SUBAPPLICATION Uebung_002a5b_AX (* DigitalInput_I1-3 mit OR auf DigitalOutput_Q1-3, mit Plug and Socket *)
  (* Standard: 61499-2; Description: Copyright (c) 2023 Meisterschulen am Ostbahnhof This program and the accompanying materials are made available under the terms of the Eclipse Public License 2.0 which is available at https://www.eclipse.org/legal/epl-2.0/ SPDX-License-Identifier: EPL-2.0 *)
  (* Version 1.0, 2023-10-23, Franz Höpfinger, Meisterschulen am Ostbahnhof, initial API and implementation and/or initial documentation *)
  PACKAGE Uebungen;
  IMPORT logiBUS::io::DI::logiBUS_DI::Input_I1;
  IMPORT logiBUS::io::DI::logiBUS_DI::Input_I2;
  IMPORT logiBUS::io::DI::logiBUS_DI::Input_I3;
  IMPORT logiBUS::io::DQ::logiBUS_DO::Output_Q1;
  IMPORT logiBUS::io::DQ::logiBUS_DO::Output_Q2;
  IMPORT logiBUS::io::DQ::logiBUS_DO::Output_Q3;
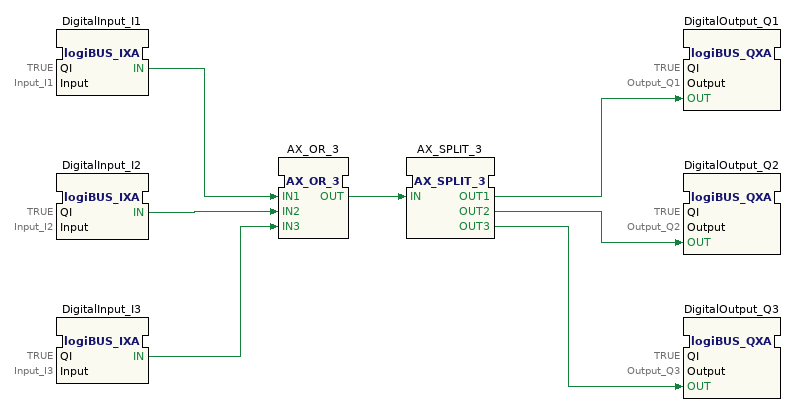
  FBS
    DigitalInput_I1 : logiBUS::io::DI::logiBUS_IXA(QI := TRUE, Input := Input_I1);
    DigitalOutput_Q1 : logiBUS::io::DQ::logiBUS_QXA(QI := TRUE, Output := Output_Q1);
    AX_OR_3 : adapter::booleanOperators::AX_OR_3;
    DigitalInput_I2 : logiBUS::io::DI::logiBUS_IXA(QI := TRUE, Input := Input_I2);
    DigitalInput_I3 : logiBUS::io::DI::logiBUS_IXA(QI := TRUE, Input := Input_I3);
    DigitalOutput_Q2 : logiBUS::io::DQ::logiBUS_QXA(QI := TRUE, Output := Output_Q2);
    DigitalOutput_Q3 : logiBUS::io::DQ::logiBUS_QXA(QI := TRUE, Output := Output_Q3);
    AX_SPLIT_3 : adapter::events::unidirectional::AX_SPLIT_3;
  END_FBS
  ADAPTER_CONNECTIONS
    DigitalInput_I1.IN TO AX_OR_3.IN1;
    DigitalInput_I2.IN TO AX_OR_3.IN2;
    DigitalInput_I3.IN TO AX_OR_3.IN3;
    AX_OR_3.OUT TO AX_SPLIT_3.IN;
    AX_SPLIT_3.OUT1 TO DigitalOutput_Q1.OUT;
    AX_SPLIT_3.OUT2 TO DigitalOutput_Q2.OUT;
    AX_SPLIT_3.OUT3 TO DigitalOutput_Q3.OUT;
  END_CONNECTIONS
END_SUBAPPLICATION
